{attribute 'qualified_only'}
{attribute 'strict'}
TYPE E_AccessType :
(
	READ,
	WRITE,
	READWRITE
);
END_TYPE

(* stored: Version 1.1.0.1, ProductVersion 3.1.4024.12
   DUT E_AccessType: Id {3b4a0574-58fe-4887-976d-331b582e641f} *)
